(* CoDeSys 2.3.9.37 project: Cap10_1.pro *)
(* Libraries: STANDARD.LIB 4.10.05 12:14:46 *)

(* Global variable list: Globale_Variablen *)
VAR_GLOBAL

	(*Entradas*)
	Start : BOOL;
	ControlOK : BOOL;

      (*Salidas*)
	Warning : BOOL;
	Stop : BOOL;
END_VAR

(* POU PLC_PRG, FBD *)
PROGRAM PLC_PRG
VAR

END_VAR
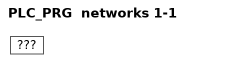
_FBD_ (* Function Block Diagram *)
NETWORK 1
	???
_END_FBD_
(* the same logic as Structured Text *)
(* Network 1 *)
END_PROGRAM

(* Visualisation Observation
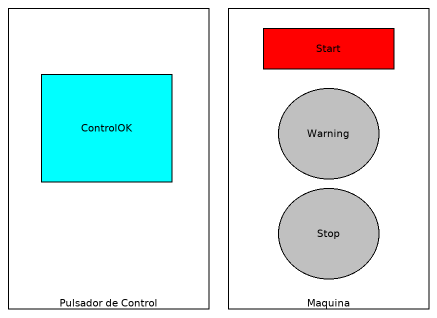
rectangle at (230,10)-(431,311): text "Maquina"
rectangle at (10,10)-(211,311): text "Pulsador de Control"
rectangle at (43,76)-(174,184): text "ControlOK"; alarm colour if ControlOK; toggles ControlOK
ellipse at (280,90)-(381,181): text "Warning"; alarm colour if Warning
ellipse at (280,190)-(381,281): text "Stop"; alarm colour if Stop
rectangle at (265,30)-(396,71): text "Start"; alarm colour if Start; toggles Start
*)
